{attribute 'qualified_only'}
{attribute 'strict'}
TYPE EjectionGateMode :
(
	Mode_Standard	:= 0,
	Mode_Manual		:= 1,
	Mode_Simulation	:= 2
	
);
END_TYPE

(* stored: Version 1.1.0.1, ProductVersion 3.1.4024.12
   DUT EjectionGateMode: Id {dd55af88-da98-4111-b1d7-3877a54d9411} *)
